// TwinCAT 3 PLC project Project_Logic
// Title: Project_Logic_1
// Company: InTimeTec
// ProjectVersion: 0.1.0.1
// ProgramVersion: 3.1.4024.0
// libraries:
//   Tc2_Standard, * (Beckhoff Automation GmbH)
//   Tc2_System, * (Beckhoff Automation GmbH)
//   Tc3_Module, * (Beckhoff Automation GmbH)
// project tree:
//   / PlcTask.TcTTO
//   POUs/ FB_BottleFiller.TcPOU, MAIN.TcPOU
//   Version/ Global_Version.TcGVL
// (motion and I/O tree: see PLC project test_project)
// real-time tasks:
//   TASK PlcTask: cycle T#10ms, priority 20, ADS port 350
//   TASK PlcTask1: cycle T#10ms, priority 21, ADS port 351

CONFIGURATION Project_Logic
    RESOURCE PLC ON TwinCAT3
        TASK PlcTask(INTERVAL := T#10ms, PRIORITY := 21);
        PROGRAM MAIN WITH PlcTask : MAIN;
    END_RESOURCE
END_CONFIGURATION

// ---- Version/Global_Version.TcGVL
{attribute 'TcGenerated'}
{attribute 'no-analysis'}
{attribute 'linkalways'}
// This function has been automatically generated from the project information.
VAR_GLOBAL CONSTANT
	{attribute 'const_non_replaced'}
	stLibVersion_Project_Logic_1 : ST_LibVersion := (iMajor := 0, iMinor := 1, iBuild := 0, iRevision := 1, nFlags := 0, sVersion := '0.1.0.1');
END_VAR

// ---- POUs/MAIN.TcPOU
PROGRAM MAIN
VAR
	fbBottle : FB_BottleFiller;
END_VAR

fbBottle.StartFilling();

END_PROGRAM

// ---- POUs/FB_BottleFiller.TcPOU
FUNCTION_BLOCK FB_BottleFiller
VAR_INPUT
	bLevelSensor : BOOL;
END_VAR
VAR
	bFillingValve : BOOL;
	bValvePressure : DINT ;
	bisTankEmpty : BOOL;
END_VAR
VAR_OUTPUT
	bFilling : BOOL;
	bSpeed : DINT;
END_VAR

METHOD SetValvePressure
VAR_INPUT
	bPressureValue : DINT;
END_VAR
bValvePressure := bPressureValue;
bSpeed := bValvePressure -10;
END_METHOD

METHOD StartFilling : BOOL
VAR_INPUT
END_VAR
IF bisTankEmpty THEN
	bFilling := bFillingValve := TRUE;
	
END_IF
END_METHOD

METHOD StopFilling : BOOL
VAR_INPUT
END_VAR
IF bLevelSensor THEN
	bFilling := bFillingValve := FALSE;
END_IF
END_METHOD

END_FUNCTION_BLOCK
